FUNCTION_BLOCK PAEActValve EXTENDS PAEActuator1way
VAR_INPUT
END_VAR
VAR_OUTPUT
END_VAR
VAR
END_VAR

METHOD PUBLIC PAEActValve
VAR_INPUT
END_VAR
END_METHOD

END_FUNCTION_BLOCK

(* stored: Version 1.1.0.1, ProductVersion 3.1.4020.12
   POU PAEActValve: Id {2e9e0893-b9af-4ab8-aa78-98b7c83fff2e}, SpecialFunc None
   Method PAEActValve: Id {ddcd5fdd-00ef-469d-8539-11dca43d9b15} *)
